(* IEC 61131-3 sources: eCockpitGit/test_project/src/%F%00 Library/%F%Common Functions/%F%Buffer/%POU%FB_FIFOArray/%PRO%isNotEmpty, 1 file *)

(* ---- %GETSET%Get.st ---- *)
//Returns wether the buffer is not empty
// |**Version**|**Author**| **Date** |**Changes**
// | 1         | NSN      | 15-02-22 | Creation
VAR
END_VAR

(*%!%__DELIMITER__%!%*)
isNotEmpty		:=		S_amount > 0;
